// TIA Portal V17 export
// export: Created 2024-08-29T18:23:50.1459397Z, ExportSetting WithDefaults, DisplayName Totally Integrated Automation Portal, DisplayVersion V17 Update 7, DisplayName TIA Portal Openness, DisplayVersion V17 Update 7, DisplayName TIA Portal Version Control Interface, DisplayVersion V17, DisplayName SINAMICS Startdrive Advanced, DisplayVersion V17 SP2, DisplayName SINAMICS Startdrive G110M, G120, G120C, G120D, G120P, G115D, DisplayVersion V17 SP2, DisplayName SINAMICS Startdrive G130, G150, S120, S150, SINAMICS MV, S210, DisplayVersion V17 SP2, DisplayName STEP 7 Professional, DisplayVersion V17 Update 7, DisplayName STEP 7 Safety, DisplayVersion V17 Update 6, DisplayName WinCC Advanced / Unified PC, DisplayVersion V17 Update 7
VAR_GLOBAL   // PLC tag table "digitalFielbusOutputs"
   qCylinder1DirectionA AT %Q149.0 : Bool;
   qCylinder1DirectionB AT %Q151.0 : Bool;
   qCylinder2DirectionA AT %Q149.1 : Bool;
   qCylinder2DirectionB AT %Q151.1 : Bool;
   qCylinder7DirectionA AT %Q149.6 : Bool;
   qCylinder7DirectionB AT %Q151.6 : Bool;
   qCylinder4DirectionA AT %Q149.3 : Bool;
   qCylinder4DirectionB AT %Q151.3 : Bool;
   qCylinder5DirectionA AT %Q149.4 : Bool;
   qCylinder5DirectionB AT %Q151.4 : Bool;
   qCylinder6DirectionA AT %Q149.5 : Bool;
   qCylinder6DirectionB AT %Q151.5 : Bool;
   qCylinder3DirectionA AT %Q149.2 : Bool;
   qCylinder3DirectionB AT %Q151.2 : Bool;
   qCylinder8DirectionA AT %Q149.7 : Bool;
   qCylinder8DirectionB AT %Q151.7 : Bool;
   qCylinder9DirectionA AT %Q148.0 : Bool;
   qCylinder9DirectionB AT %Q150.0 : Bool;
   qCylinder10DirectionA AT %Q148.1 : Bool;
   qCylinder10DirectionB AT %Q150.1 : Bool;
   qActivateCutOffValve AT %Q147.0 : Bool;
END_VAR
